// Mitsubishi GX Works2 project: 세탁기   PLC: Q03UDV

PROGRAM MAIN
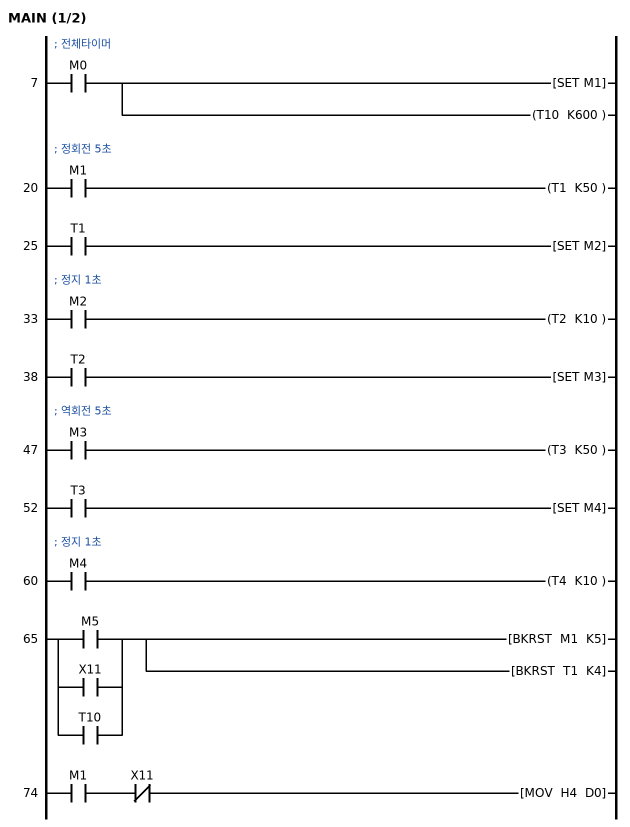
; 전체타이머
7     LD      M0
      SET     M1
      OUT     T10 K600
; 정회전 5초
20    LD      M1
      OUT     T1 K50
25    LD      T1
      SET     M2
; 정지 1초
33    LD      M2
      OUT     T2 K10
38    LD      T2
      SET     M3
; 역회전 5초
47    LD      M3
      OUT     T3 K50
52    LD      T3
      SET     M4
; 정지 1초
60    LD      M4
      OUT     T4 K10
65    LD      M5
      OR      X11
      OR      T10
      BKRST   M1 K5
      BKRST   T1 K4
74    LD      M1
      ANI     X11
      MOV     H4 D0
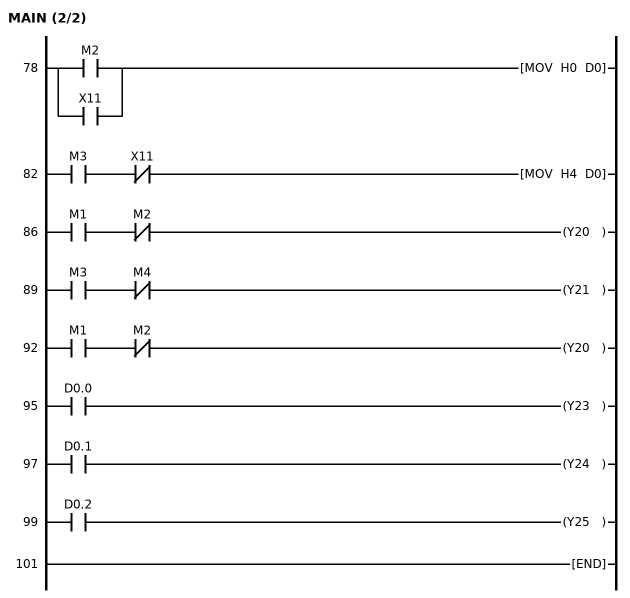
78    LD      M2
      OR      X11
      MOV     H0 D0
82    LD      M3
      ANI     X11
      MOV     H4 D0
86    LD      M1
      ANI     M2
      OUT     Y20
89    LD      M3
      ANI     M4
      OUT     Y21
92    LD      M1
      ANI     M2
      OUT     Y20
95    LD      D0.0
      OUT     Y23
97    LD      D0.1
      OUT     Y24
99    LD      D0.2
      OUT     Y25
101   END
END_PROGRAM
